(* IEC 61131-3 sources: verifaps-lib/aps-rvt/src/test/resources, 4 files *)

(* ---- caseif_new.st ---- *)
PROGRAM abc
VAR_INPUT  i : INT; END_VAR
VAR_OUTPUT o : INT; END_VAR

CASE i OF
  0:        o := 0;
  1..5:     o := i * i;
  5..10:    o := i+(i*2);
  ELSE      o := -1;
END_CASE

END_PROGRAM

(* ---- caseif_old.st ---- *)
PROGRAM abc
VAR_INPUT  i : INT; END_VAR
VAR_OUTPUT o : INT; END_VAR

IF i = 0 THEN
    o := 0;
ELSEIF i > 0 AND i <= 5 THEN
    o := i * i;
ELSEIF i > 4 AND i <= 10 THEN
    o := i+i*2;
ELSE
    o := -1;
END_IF

END_PROGRAM

(* ---- simple1_new.st ---- *)
PROGRAM abc
VAR_INPUT i : INT; END_VAR
VAR_OUTPUT o : INT; END_VAR
o:= 2*i;
END_PROGRAM

(* ---- simple1_old.st ---- *)
PROGRAM abc
VAR_INPUT i : INT; END_VAR
VAR_OUTPUT o : INT; END_VAR
o:= i+i;
END_PROGRAM
